// TIA Portal V20 export
TYPE "typeEm1MonitoringCmStatus"
// stored: Access Published, Namespace Unit1
   STRUCT
      uwAxisB { ExternalWritable := 'False'} : "LBC_typeAxisControlNodeMonitoring";
      airShaft { ExternalWritable := 'False'} : "LBC_typeTwoWayActuatorControlNodeMonitoring";
      expel { ExternalWritable := 'False'} : "LBC_typeTwoWayActuatorControlNodeMonitoring";
      tensionSnr { ExternalWritable := 'False'} : "LBC_typeDigitalSignalControlNodeMonitoring";
      radius { ExternalWritable := 'False'} : "LBC_typeAnalogInputControlNodeMonitoring";
   END_STRUCT;
END_TYPE
